SUBAPPLICATION Uebung_080b (* Beispiel für E_CTU mit E_SPLIT für Event-Verdoppelung *)
  (* Standard: 61499-2; Description: Copyright (c) 2023 Meisterschulen am Ostbahnhof This program and the accompanying materials are made available under the terms of the Eclipse Public License 2.0 which is available at https://www.eclipse.org/legal/epl-2.0/ SPDX-License-Identifier: EPL-2.0 Beispiel für E_CTU Aufwärts zählen UAO Curriculum Module 3 - The IEC 61499 Standard, Seite 92 *)
  (* Version 1.0, 2023-10-23, Franz Höpfinger, Meisterschulen am Ostbahnhof *)
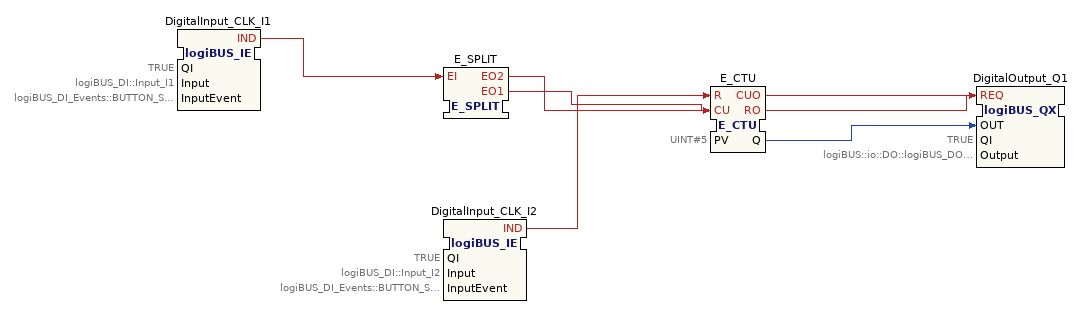
  (* E_SPLIT macht 2 Events, die dann wieder gemerged werden. --> Event wird verdoppelt *)
  FBS
    DigitalOutput_Q1 : logiBUS_QX(QI := TRUE, Output := logiBUS::io::DO::logiBUS_DO::Output_Q1);
    DigitalInput_CLK_I1 : logiBUS_IE(QI := TRUE, Input := logiBUS_DI::Input_I1, InputEvent := logiBUS_DI_Events::BUTTON_SINGLE_CLICK);
    E_CTU : E_CTU(PV := UINT#5);
    DigitalInput_CLK_I2 : logiBUS_IE(QI := TRUE, Input := logiBUS_DI::Input_I2, InputEvent := logiBUS_DI_Events::BUTTON_SINGLE_CLICK);
    E_SPLIT : E_SPLIT;
  END_FBS
  EVENT_CONNECTIONS
    E_CTU.CUO TO DigitalOutput_Q1.REQ;
    E_CTU.RO TO DigitalOutput_Q1.REQ;
    DigitalInput_CLK_I2.IND TO E_CTU.R;
    E_SPLIT.EO2 TO E_CTU.CU;
    DigitalInput_CLK_I1.IND TO E_SPLIT.EI;
    E_SPLIT.EO1 TO E_CTU.CU;
  END_CONNECTIONS
  DATA_CONNECTIONS
    E_CTU.Q TO DigitalOutput_Q1.OUT;
  END_CONNECTIONS
END_SUBAPPLICATION
